PROGRAM P_HMI
VAR
	fDelta: LREAL;
	fbStats: FB_STATS;
	bZerarGraficoHMI: BOOL;
END_VAR

(* Actual Validation Values on FB_WEIGHING Block*)

GVL_WEIGHING_HMI.nActualWindowLenght 					 	:= MAIN.fbDynamicWeighing.nActualWindowLenght;


(* Validation *)
GVL_WEIGHING_HMI.nActualValidationSamplesValidation		 	:= MAIN.fbDynamicWeighing.nActualValidationSamplesValidation;
GVL_WEIGHING_HMI.fActualThresholdWeightValidation 		 	:= MAIN.fbDynamicWeighing.fActualThresholdWeightValidation;
GVL_WEIGHING_HMI.fActualMaxStdValidation					:= MAIN.fbDynamicWeighing.fActualMaxStdValidation;
GVL_WEIGHING_HMI.fActualMaxWeightDeviationValidation		:= MAIN.fbDynamicWeighing.fActualMaxWeightDeviationValidation;
GVL_WEIGHING_HMI.fActualRelativeWeightLimit					:= MAIN.fbDynamicWeighing.fActualRelativeWeightLimit;

(* AutoTare*)

GVL_WEIGHING_HMI.nActualValidationSamplesAutoTare			:= MAIN.fbDynamicWeighing.nActualValidationSamplesAutoTare;
GVL_WEIGHING_HMI.fActualThresholdWeightAutoTare 			:= MAIN.fbDynamicWeighing.fActualThresholdWeightAutoTare;
GVL_WEIGHING_HMI.fActualMaxStdAutoTare						:= MAIN.fbDynamicWeighing.fActualMaxStdAutoTare;
GVL_WEIGHING_HMI.fActualMaxWeightDeviationAutoTare			:= MAIN.fbDynamicWeighing.fActualMaxWeightDeviationAutoTare;
	
GVL_WEIGHING_HMI.fWeight 									:= MAIN.fbDynamicWeighing.fWeight;
GVL_WEIGHING_HMI.fLastWeight 								:= MAIN.fbDynamicWeighing.fLastWeight;
GVL_WEIGHING_HMI.fStd 										:= MAIN.fbDynamicWeighing.fStd;
GVL_WEIGHING_HMI.fLastStd 									:= MAIN.fbDynamicWeighing.fLastStd;


(* Booleans *)

GVL_WEIGHING_HMI.bValidMeasurement 	:= MAIN.fbDynamicWeighing.bValidMeasurement;
GVL_WEIGHING_HMI.bNewResult			:= MAIN.fbDynamicWeighing.bNewResult;

(* Auto Reset Reconfigure Bits *)
IF GVL_WEIGHING_HMI.bReconfigureWeighing THEN
	GVL_WEIGHING_HMI.bReconfigureWeighing := FALSE;
END_IF


(* Bit for Criterias Management *)
IF MAIN.fbDynamicWeighing.fWeight > MAIN.fbDynamicWeighing.fActualThresholdWeightValidation THEN
	GVL_WEIGHING_HMI.bCriteria1 := TRUE;
	fDelta := MAIN.fbDynamicWeighing.fMax - MAIN.fbDynamicWeighing.fMin;	
	IF MAIN.fbDynamicWeighing.fMax - MAIN.fbDynamicWeighing.fMin 
		< MAIN.fbDynamicWeighing.fActualMaxWeightDeviationValidation THEN
			GVL_WEIGHING_HMI.bCriteria2 := TRUE;
		IF MAIN.fbDynamicWeighing.fStd < MAIN.fbDynamicWeighing.fActualMaxStdValidation THEN
			GVL_WEIGHING_HMI.bCriteria3 := TRUE;
		END_IF
	END_IF
ELSE (* Reset everytime weight is < than threshold *)
	GVL_WEIGHING_HMI.bCriteria1 := FALSE;
	GVL_WEIGHING_HMI.bCriteria2 := FALSE;
	GVL_WEIGHING_HMI.bCriteria3	:= FALSE;
END_IF


(* Stats *)
fbStats(
	bValidMeasurement:= MAIN.fbDynamicWeighing.bValidMeasurement, 
	fLastWeight:= MAIN.fbDynamicWeighing.fLastWeight, 
	fLastStd:= MAIN.fbDynamicWeighing.fLastStd, 
	bNewResult:= MAIN.fbDynamicWeighing.bNewResult, 
	bZerarGrafico:= bZerarGraficoHMI,
	fReferenceMeasurement:= MAIN.aRawSignal[1], 
	fMaxWeight=> , 
	fMinWeight=> , 
	fDelta=> , 
	fMinReference=> , 
	fMaxReference=> , 
	fDeltaReference=> );


(* FB_Scale Diag *)
GVL_WEIGHING_HMI.bFbScaleCfgd := MAIN.fbDynamicWeighing.fbScaleCfgBit;
GVL_WEIGHING_HMI.bFbScaleCfgd := MAIN.fbDynamicWeighing.fbScaleCfgBit;
GVL_WEIGHING_HMI.eFbScaleState	:= MAIN.fbDynamicWeighing.fbScaleEnumState;

END_PROGRAM

(* stored: Version 1.1.0.1, ProductVersion 3.1.4026.17
   POU P_HMI: Id {23683a70-86f5-4b64-ba26-edc9c2b44b03}, SpecialFunc None *)
